{attribute 'GeneratedUsingTerminal: EL2521-0000-1019'}
{attribute addProperty BoxType "EL2521-0000-1019"}
{attribute addProperty Description "EL2521 1Ch. Pulse Train Output"}
{attribute addProperty Physics "KK"}
{attribute addProperty Id "PTO_StatusAT %I*PTO_Status_40B3051C7ENC_Status_compactAT %I*ENC_Status_compact_036460C97PTO_ControlAT %Q*PTO_Control_9287F8E45PTO_Target_compactAT %Q*PTO_Target_compact_5C359F7D2ENC_Control_compactAT %Q*ENC_Control_compact_2ED727EF3WcStateAT %I*WcState_9091E0EB2InfoDataAT %I*InfoData_32EB74EA10"}
{attribute addProperty CRC "131800045"}
{attribute addProperty Size "36"}
TYPE EL2521_07DB1BED EXTENDS EtcSlaveTerminalBase_947E5A46 :
STRUCT
	{attribute addProperty Name "PTO_Status"}
	PTO_Status : PTO_Status_40B3051C;
	{attribute addProperty Name "ENC_Status_compact"}
	ENC_Status_compact : ENC_Status_compact_036460C9;
	{attribute addProperty Name "PTO_Control"}
	PTO_Control : PTO_Control_9287F8E4;
	{attribute addProperty Name "PTO_Target_compact"}
	PTO_Target_compact : PTO_Target_compact_5C359F7D;
	{attribute addProperty Name "ENC_Control_compact"}
	ENC_Control_compact : ENC_Control_compact_2ED727EF;
	{attribute addProperty Name "WcState"}
	WcState : WcState_9091E0EB;
	{attribute addProperty Name "InfoData"}
	InfoData : InfoData_32EB74EA;
END_STRUCT
END_TYPE

(* stored: Version 1.2.0.0, ProductVersion 3.1.4024.9
   DUT EL2521_07DB1BED: Id {f14cf39c-17ea-44e5-8b27-9caf2bd5dd08} *)
